INTERFACE ITF_SITP_PolecenieZmianyStanu EXTENDS ITF_SITP_PolecenieZmiany

METHOD PUBLIC zwrocRodzajPolecenia : E_SITP_PolecenieZmianyStanu
VAR_INPUT
END_VAR
END_METHOD

END_INTERFACE

(* stored: Version 1.1.0.1
   Itf ITF_SITP_PolecenieZmianyStanu: Id {1080afa1-981a-0963-2622-1fa15f0d99ff}
   Method zwrocRodzajPolecenia: Id {0005fcad-4874-005f-2c98-d0503e9bdf1c} *)
